INTERFACE INTERNAL _I_ValidateGeneric EXTENDS __SYSTEM.IQueryInterface, I_Debug

END_INTERFACE

(* stored: Version 1.1.0.1
   Itf _I_ValidateGeneric: Id {2485e777-bc34-4faa-9644-c49ae0e559ef} *)
